PROGRAM POU
VAR
	fbtimer1:TOF;
	rs:RS;
	BLINK1 :BLINK;
	TIMELOW:TIME;
	Initialschritt:SR;
	Schritt1:SR;
	Schritt2:SR;
	Schritt3:SR;
	Schritt4:SR;
	Schritt5:SR;

	
	
END_VAR

VAR_INPUT
	i3 AT %I*:BOOL;
	i4 AT %I*:BOOL;
	i5 AT %I*:BOOL;
	i6 AT %I*:BOOL;
	i7 AT %I*:BOOL;
END_VAR
VAR_OUTPUT
	a2 AT %Q*: BOOL;
	a3 AT %Q*: BOOL;
	a4 AT %Q*: BOOL;
	a5 AT %Q*: BOOL;
	a6 AT %Q*: BOOL;
	a7 AT %Q*: BOOL;
	a8 AT %Q*: BOOL;
END_VAR

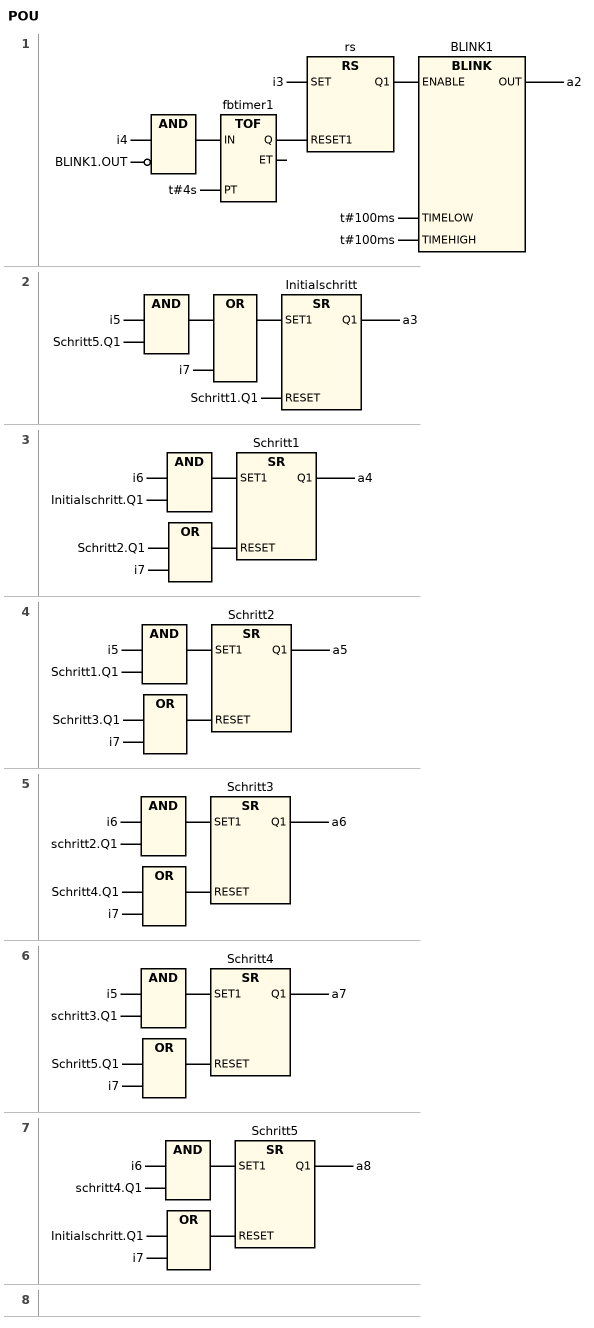
// NETWORK 1
fbtimer1(IN := i4 AND NOT BLINK1.OUT, PT := t#4s); // TOF
rs(SET := i3, RESET1 := fbtimer1.Q);
BLINK1(ENABLE := rs.Q1, TIMELOW := t#100ms, TIMEHIGH := t#100ms); // BLINK
a2 := BLINK1.OUT;

// NETWORK 2
Initialschritt(SET1 := i5 AND Schritt5.Q1 OR i7, RESET := Schritt1.Q1); // SR
a3 := Initialschritt.Q1;

// NETWORK 3
Schritt1(SET1 := i6 AND Initialschritt.Q1, RESET := Schritt2.Q1 OR i7); // SR
a4 := Schritt1.Q1;

// NETWORK 4
Schritt2(SET1 := i5 AND Schritt1.Q1, RESET := Schritt3.Q1 OR i7); // SR
a5 := Schritt2.Q1;

// NETWORK 5
Schritt3(SET1 := i6 AND schritt2.Q1, RESET := Schritt4.Q1 OR i7); // SR
a6 := Schritt3.Q1;

// NETWORK 6
Schritt4(SET1 := i5 AND schritt3.Q1, RESET := Schritt5.Q1 OR i7); // SR
a7 := Schritt4.Q1;

// NETWORK 7
Schritt5(SET1 := i6 AND schritt4.Q1, RESET := Initialschritt.Q1 OR i7); // SR
a8 := Schritt5.Q1;

// NETWORK 8

END_PROGRAM

(* stored: Version 1.1.0.1, ProductVersion 3.1.4024.4
   POU POU: Id {7a78f167-2b48-4c2c-bd55-ecaf2418a337}, SpecialFunc None *)
